FUNCTION_BLOCK FB_HSSController IMPLEMENTS I_HydraulicMixingControl
VAR_INPUT
END_VAR
VAR_OUTPUT
END_VAR
VAR
	//Properties
	bError 			: BOOL 				:= FALSE;
	eMode 			: E_ControlMode 	:= E_ControlMode.Off;
	ePumpMode 		: E_PumpControlMode := E_PumpControlMode.OFF;
	fPumpSet 		: REAL 				:= 0;
	fTemperatureAct : REAL              := 18;
	fTemperatureSet : REAL				:= 45;
	fValveSet 		: REAL 				:= 0;
	
	//PID
	fbPID : FB_PID; //Set PID parameters (Kp, Ti, ...) in Auto method
	
	//Manual mode
	eManualPumpMode	: E_PumpControlMode := E_PumpControlMode.NONE;
	fManualPumpSet	: REAL 				:= fPumpSet;
	fManualValveSet : REAL 				:= fValveSet;
	
END_VAR

METHOD Auto
VAR
	//PID params
	Kp		:	REAL	:=	1.4;	//Proportional gain
	Ti		:	REAL	:=	80;		//Integral time
	Td		:	REAL	:=	0;		//Derivative time
	LimLow	:	REAL	:=	0;		//Low limit of output
	LimHigh	:	REAL	:=	100;	//High limit of output
	bReverseActing	:	BOOL := FALSE;
	
	//Heating Curve
	fSlope	: 	REAL	:= 	-1.0;
	fOffset	: 	REAL	:= 	45.0;
END_VAR
//TROX controls heating power via throttle circuit
//Calculate supply water set temperature from heating curve, 45 °C at 0 °C ambient temperature

fTemperatureSet := FC_HeatingCurve(	fTempAmb := GVL.fTempAmbAir,
									fSlope := fSlope,
									fOffset := fOffset);

//PID control for valve
fbPID(
	xSet:= fTemperatureSet, 
	xAct:= fTemperatureAct, 
	Kp:= Kp, 
	Ti:= Ti, 
	Td:= Td, 
	LimLow:= LimLow, 
	LimHigh:= LimHigh, 
	bReverseActing:= bReverseActing, 
	RST:= FALSE, 
	Y=> fValveSet
	);

//Pump setpoint just constant for now
fPumpSet 	:= 60; //60 % of nominal power
ePumpMode 	:= E_PumpControlMode.CONST_DIFFPRESS;
END_METHOD

PROPERTY Error : BOOL
GET
Error := THIS^.bError;
END_GET
SET
THIS^.bError := Error;
END_SET
END_PROPERTY

METHOD ExternalADSControl
VAR_INPUT
END_VAR
//Set Valve position according to ADS command
fValveSet := ADS.fHSSValveSetADS;

//Set pump operation and set point to ADS command
fPumpSet 	:= ADS.fHSSPumpSetpointADS; // % of nominal power
ePumpMode 	:= ADS.eHSSPumpContModeADS;
END_METHOD

{warning 'add method implementation '}
METHOD Init : BOOL
END_METHOD

METHOD Manual
ePumpMode 	:= eManualPumpMode;
fPumpSet 	:= fManualPumpSet;
fValveSet 	:= fManualValveSet;
END_METHOD

PROPERTY Mode : E_ControlMode
GET
Mode := THIS^.eMode;
END_GET
SET
THIS^.eMode := Mode;
END_SET
END_PROPERTY

METHOD Off
fPumpSet	:=	0;
ePumpMode	:=	E_PumpControlMode.OFF;
fValveSet 	:=	0;
END_METHOD

{warning 'add method implementation '}
METHOD OperationTest : BOOL
END_METHOD

PROPERTY PumpMode : E_PumpControlMode
GET
PumpMode := THIS^.ePumpMode;
END_GET
SET
THIS^.ePumpMode := PumpMode;
END_SET
END_PROPERTY

PROPERTY PumpSet : REAL
GET
PumpSet := THIS^.fPumpSet;
END_GET
SET
THIS^.fPumpSet := PumpSet;
END_SET
END_PROPERTY

METHOD Run
//Run control routine according to mode set
CASE eMode OF
	E_ControlMode.Off:		   			Off();
	E_ControlMode.Init:		   			Init();
	E_ControlMode.OperationTest:	    OperationTest();
	E_ControlMode.Auto:   				Auto();
	E_ControlMode.Manual:				Manual();
	E_ControlMode.ExternalADSControl:	ExternalADSControl();
END_CASE

//Write temperature supply setpoint to GVL
GVL.fHSSTempSupSet := THIS^.TemperatureSupSet;
END_METHOD

PROPERTY TemperatureSupAct : REAL
GET
TemperatureSupAct := THIS^.fTemperatureAct;
END_GET
SET
THIS^.fTemperatureAct := TemperatureSupAct;
END_SET
END_PROPERTY

PROPERTY TemperatureSupSet : REAL
GET
TemperatureSupSet := THIS^.fTemperatureSet;
END_GET
SET
THIS^.fTemperatureSet := TemperatureSupSet;
END_SET
END_PROPERTY

PROPERTY ValveSet : REAL
GET
ValveSet := THIS^.fValveSet;
END_GET
SET
THIS^.fValveSet := ValveSet;
END_SET
END_PROPERTY

END_FUNCTION_BLOCK

(* stored: Version 1.1.0.1, ProductVersion 3.1.4024.3
   POU FB_HSSController: Id {048ccbd4-7cc8-4766-ac9c-957fc8886059}, SpecialFunc None
   Method Auto: Id {583c682a-938e-4181-98c5-029b87793184}
   Property Error: Id {180141a3-3cf2-45cf-9e99-4a8eef933947}
   Get Get: Id {4bd89ef3-ee54-489b-8d94-8a87a7b8043c}
   Set Set: Id {714c0069-575c-4c6f-bc78-122738092186}
   Method ExternalADSControl: Id {357d61c9-1b6c-4126-969f-606af2eba9d5}
   Method Init: Id {8a22dabf-7d63-456f-b1c1-b275299923ac}
   Method Manual: Id {25e4144a-b453-44b7-a3eb-5ddb8b7b4501}
   Property Mode: Id {163be683-95ac-4ed0-8631-30e429c6e96c}
   Get Get: Id {73d6d545-3fdb-4bfa-9eb4-6bf9b7ff45a5}
   Set Set: Id {3045bf94-5c9a-4203-bbb1-0c8deda7e4eb}
   Method Off: Id {5e246dea-33fd-446a-8df7-4a4bd250c053}
   Method OperationTest: Id {fa6e2932-63a5-4e65-b417-dc0aaa4d4bcc}
   Property PumpMode: Id {0a436de6-a19e-4c0c-b426-cf524e061545}
   Get Get: Id {b373e47a-5046-4b72-8648-bf7a07d972f3}
   Set Set: Id {b4b1c6f4-bd41-4cb7-bb02-09ea2f4fa04b}
   Property PumpSet: Id {dca9e9f8-dcad-4d11-9a47-00a61b59f42f}
   Get Get: Id {1a87bc90-cd31-41fb-b0c2-8ebaf870c7c2}
   Set Set: Id {ea81d5d1-f3d8-4fb6-a93f-8dc9750ce396}
   Method Run: Id {cc816fbe-aca6-4acb-9b51-3927954539ff}
   Property TemperatureSupAct: Id {9de2feb8-f0be-4aa6-8f93-c7cb522d7a15}
   Get Get: Id {3df50ce9-44b0-49ff-ba39-70ed9b8485bd}
   Set Set: Id {301194e1-b939-4ce9-8461-fe6af9a53234}
   Property TemperatureSupSet: Id {515fdf1d-d6ed-485e-af64-9ac743bc86e4}
   Get Get: Id {ac1fdfa8-afe1-45cd-b6fb-6df60c663836}
   Set Set: Id {af7bdacb-0df8-4d36-942d-507fb97727b5}
   Property ValveSet: Id {3c8859be-1b44-46f8-a8a6-7e5fbf5bdeb1}
   Get Get: Id {4a480c83-f7e2-4927-85ec-d320ceef74d6}
   Set Set: Id {f2fba49f-c614-44ea-8cd0-bb97f3c85320} *)
